// TwinCAT 3 PLC project PLC1
// ProgramVersion: 3.1.4020.1
// libraries:
//   Tc2_Standard, * (Beckhoff Automation GmbH)
//   Tc2_System, * (Beckhoff Automation GmbH)
//   Tc3_Module, * (Beckhoff Automation GmbH)
// project tree:
//   / GlobalTextList.TcGTLO, PlcTask.TcTTO, Visualization Manager.TcVMO (not stored)
//   POUs/ MAIN.TcPOU
//   VISUs/ Visualization.TcVIS
// real-time tasks:
//   TASK PlcTask: cycle T#10ms, priority 20, ADS port 350

CONFIGURATION PLC1
    RESOURCE PLC ON TwinCAT3
        TASK PlcTask(INTERVAL := T#10ms, PRIORITY := 20);
        PROGRAM MAIN WITH PlcTask : MAIN;
    END_RESOURCE
END_CONFIGURATION

// ---- POUs/MAIN.TcPOU
PROGRAM MAIN
VAR
	bPizzaInOven : BOOL;
	fbMyTimer	 : TON;
	fbMyTrigger_RTRIG : R_TRIG;
	bBuzzer 	 : BOOL;
	iTotalPizzasCooked	: UDINT;
END_VAR

fbMyTimer(IN:=bPizzaInOven,PT := T#3S);

bBuzzer := fbMyTimer.Q;

fbMyTrigger_RTRIG(clk:=fbMyTimer.Q);

IF fbMyTrigger_RTRIG.Q THEN
	iTotalPizzasCooked := iTotalPizzasCooked + 1;
END_IF

END_PROGRAM

// ---- GlobalTextList.TcGTLO
TEXTLIST GlobalTextList
  3 = 'Buzzer'
  2 = 'Elapsed Time: %s'
  0 = 'Insert Pizza'
  1 = 'Remove Pizza'
END_TEXTLIST

// ---- VISUs/Visualization.TcVIS
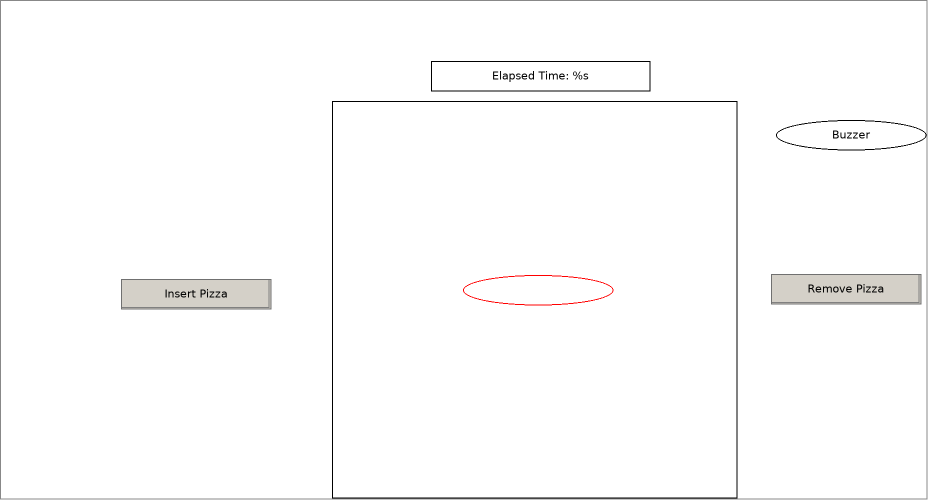
VISUALIZATION Visualization  // 928x500
    Rectangle (332,101 405x397)
    Button (121,279 150x30), "Insert Pizza"
        OnMouseDown: execute { MAIN.bPizzaInOven := TRUE; }
    Button (771,274 150x30), "Remove Pizza"
        OnMouseDown: execute { MAIN.bPizzaInOven := FALSE; }
    Ellipse (463,275 150x30), invisible if: NOT MAIN.bPizzaInOven
    Rectangle (431,61 219x30), "Elapsed Time: %s", text variable: MAIN.fbMyTimer.ET
    Ellipse (776,120 150x30), "Buzzer", colour toggle: MAIN.bBuzzer
END_VISUALIZATION
